FUNCTION_BLOCK Technology EXTENDS TcoCore.TcoContext
VAR
    _processSettings     : ProcessDataManager(THIS^);
    _technologySettings  : TechnologicalDataManager(THIS^);
    _processTraceability : ProcessDataManager(THIS^);
    {attribute addProperty Name "<#AUTOMAT ALL#>"}
    _automatAllTask : TcoCore.TcoTask(THIS^);
    {attribute addProperty Name "<#GROUND ALL#>"}
    _groundAllTask : TcoCore.TcoTask(THIS^);
    _cu00x         : CU00x(THIS^);
END_VAR

METHOD AllowAutomat : BOOL
VAR_INPUT
END_VAR
AllowAutomat := TRUE;
END_METHOD

METHOD AllowGround : BOOL
VAR_INPUT
END_VAR
AllowGround := TRUE;
END_METHOD

METHOD AllowManual :  BOOL
VAR_INPUT
END_VAR
AllowManual := TRUE;
END_METHOD

PROPERTY AutomatAllTask : REFERENCE TO TcoCore.TcoTask
GET
AutomatAllTask REF= _automatAllTask;
END_GET
END_PROPERTY

METHOD ForceStepMode : BOOL
ForceStepMode := FALSE;
END_METHOD

PROPERTY GroundAllTask : REFERENCE TO TcoCore.TcoTask
GET
GroundAllTask REF= _groundAllTask;
END_GET
END_PROPERTY

(*~
	<docu>
		<summary>
			Main method of the TcoContext. This is the entry point of any control logic that belongs to this context. 
			The call of this method is ensured by calling the <c>InstanceName.Run()</c> method, and it must not be called explicitly.
			This method is abstract, and it must be overridden in derived block.
		</summary>
	</docu>
~*)
METHOD PROTECTED Main
THIS^.RtcSynchronize(true, '', 60);
_cu00x();
END_METHOD


(*~
	<docu>
		<summary>
			Called upon exit from the context. When overridden in derived class allows to execute an arbitrary logic after closing the context cycle.	
		</summary>			
	</docu>	
~*)METHOD PROTECTED OnExit
_automatAllTask.DoneWhen(TRUE);
_groundAllTask.DoneWhen(TRUE);
END_METHOD

PROPERTY ProcessSettings : REFERENCE TO ProcessDataManager
GET
ProcessSettings REF= _processSettings;
END_GET
END_PROPERTY

PROPERTY TechnologicalSettings : REFERENCE TO TechnologicalDataManager
GET
TechnologicalSettings REF= _technologySettings;
END_GET
END_PROPERTY

END_FUNCTION_BLOCK

(* stored: Version 1.1.0.1
   POU Technology: Id {20d051ba-8e3a-4d8b-9fb7-71f6957f3a63}, SpecialFunc None
   Method AllowAutomat: Id {0aa54757-4c4d-0cde-13e5-b7414e695af4}
   Method AllowGround: Id {858f08f9-14d3-065d-1aa4-279cc3111ba4}
   Method AllowManual: Id {b0df765b-d61a-0a9e-2201-2c76ce14ddcf}
   Property AutomatAllTask: Id {af39f865-7b9c-0790-2b3f-049d4170441c}
   Get Get: Id {8b138ea6-eaf2-064a-001d-c0652c900632}
   Method ForceStepMode: Id {703a4ad0-e2bf-0a26-02d9-59b6c1ce971e}
   Property GroundAllTask: Id {517b8e00-2011-0b98-35b3-4181b5529b5d}
   Get Get: Id {ac972d75-9264-065d-3fee-04e760569681}
   Method Main: Id {d1d0e200-21d1-4642-b4c8-2fd801b60f39}
   Method OnExit: Id {29dbb73f-9a28-0fe3-31dc-e1185889822b}
   Property ProcessSettings: Id {5f876a71-a280-42cf-9f33-fc8ef671f9a2}
   Get Get: Id {4cb3435a-d869-4802-9d86-6466a1c918f7}
   Property TechnologicalSettings: Id {c5ffbe54-7294-04ed-3bd7-73d2651f9af8}
   Get Get: Id {7029ad92-6154-0241-2993-9cb7de1fadac} *)
